FUNCTION F_AddTen : INT
VAR_INPUT
	j: REFERENCE TO INT	;
END_VAR
VAR
END_VAR

F_AddTen := j+10;

END_FUNCTION

(* stored: Version 1.1.0.1, ProductVersion 3.1.4024.16
   POU F_AddTen: Id {a0b0a04e-4da7-40ad-b0f0-fd6387dbfab5}, SpecialFunc None *)
